Yaskawa INFORM job: SIDE-B-UNCLAMP.JBI

/JOB
//NAME SIDE-B-UNCLAMP
///FOLDERNAME CLAMPUNCLAMP
//POS
///NPOS 0,0,0,0,0,0
//INST
///DATE 2021/08/13 07:22
///ATTR SC,RW
NOP
'**OPEN CLAMP SIDE-B**
'*********************
'OPEN CLAMP
DOUT OT#(170) OFF
DOUT OT#(169) ON
'OPEN POKEYOKE
DOUT OT#(172) OFF
DOUT OT#(171) ON
END
